Staubli VAL3: FC_InitData.pgx

program FC_InitData()
begin
  //initial data
  cls()
  userPage()
  bRb2Start=false
  bRb2Stop=true
  bRb2Ready=false
  bSychronOn=false
  bRb2Home=false
  bRb2InitOk=false
  bTxt1=false
  bTxt2=false
  bTxt3=false
  call initCmdBuf()
end
